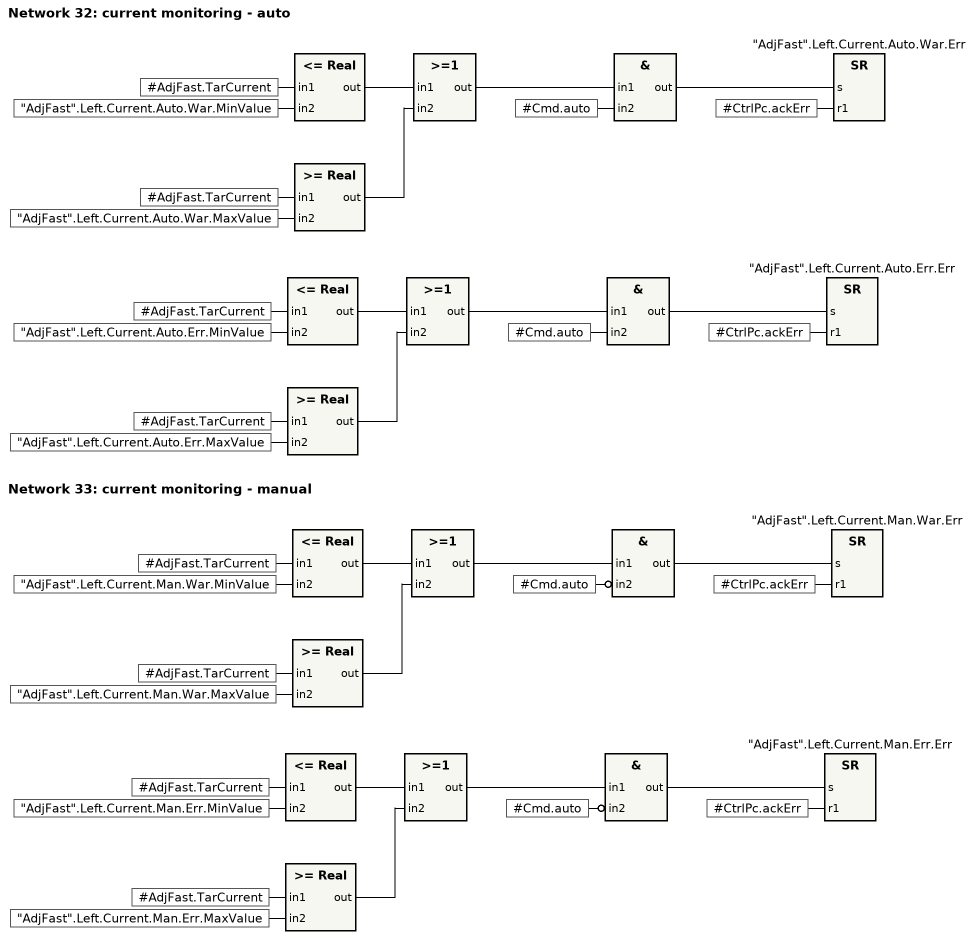
   IF ((#AdjFast.TarCurrent <= "AdjFast".Left.Current.Auto.War.MinValue) OR (#AdjFast.TarCurrent >= "AdjFast".Left.Current.Auto.War.MaxValue)) AND #Cmd.auto THEN
       "AdjFast".Left.Current.Auto.War.Err := TRUE;   // SR flip-flop
   END_IF;
   IF #CtrlPc.ackErr THEN "AdjFast".Left.Current.Auto.War.Err := FALSE; END_IF;
   IF ((#AdjFast.TarCurrent <= "AdjFast".Left.Current.Auto.Err.MinValue) OR (#AdjFast.TarCurrent >= "AdjFast".Left.Current.Auto.Err.MaxValue)) AND #Cmd.auto THEN
       "AdjFast".Left.Current.Auto.Err.Err := TRUE;   // SR flip-flop
   END_IF;
   IF #CtrlPc.ackErr THEN "AdjFast".Left.Current.Auto.Err.Err := FALSE; END_IF;
END_REGION

REGION Network 33: current monitoring - manual
   IF ((#AdjFast.TarCurrent <= "AdjFast".Left.Current.Man.War.MinValue) OR (#AdjFast.TarCurrent >= "AdjFast".Left.Current.Man.War.MaxValue)) AND NOT #Cmd.auto THEN
       "AdjFast".Left.Current.Man.War.Err := TRUE;   // SR flip-flop
   END_IF;
   IF #CtrlPc.ackErr THEN "AdjFast".Left.Current.Man.War.Err := FALSE; END_IF;
   IF ((#AdjFast.TarCurrent <= "AdjFast".Left.Current.Man.Err.MinValue) OR (#AdjFast.TarCurrent >= "AdjFast".Left.Current.Man.Err.MaxValue)) AND NOT #Cmd.auto THEN
       "AdjFast".Left.Current.Man.Err.Err := TRUE;   // SR flip-flop
   END_IF;
   IF #CtrlPc.ackErr THEN "AdjFast".Left.Current.Man.Err.Err := FALSE; END_IF;
END_REGION
END_FUNCTION_BLOCK

FUNCTION_BLOCK "AdjRight"   // FB530, FBD
{ S7_Optimized_Access := 'TRUE' }
// stored: AutoNumber false, MemoryReserve 100, SetENOAutomatically false
   VAR
      Var { ExternalAccessible := 'False'; ExternalVisible := 'False'; ExternalWritable := 'False'} : "TypeVar";
      Cmd { ExternalAccessible := 'False'; ExternalVisible := 'False'; ExternalWritable := 'False'} : "TypeCmd";
      Enc { ExternalAccessible := 'False'; ExternalVisible := 'False'; ExternalWritable := 'False'} : "SysCounterFast";
      Pos { ExternalAccessible := 'False'; ExternalVisible := 'False'; ExternalWritable := 'False'} : "SysPos";
      AdjSlow { ExternalAccessible := 'False'; ExternalVisible := 'False'; ExternalWritable := 'False'} : "SysMotor";
      AdjFast { ExternalAccessible := 'False'; ExternalVisible := 'False'; ExternalWritable := 'False'} : "SysLinMotC1150";
      TAutoOn { ExternalAccessible := 'False'; ExternalVisible := 'False'; ExternalWritable := 'False'} : TON_TIME;
      TAutoTarPosManOn { ExternalAccessible := 'False'; ExternalVisible := 'False'; ExternalWritable := 'False'} : TON_TIME;
      T { ExternalAccessible := 'False'; ExternalVisible := 'False'; ExternalWritable := 'False'} : Array[1..5] of IEC_TIMER;
      adjFastPnSlaveOff { ExternalAccessible := 'False'; ExternalVisible := 'False'; ExternalWritable := 'False'} : "SysPnSlaveDeactivate";
      tarOld { ExternalAccessible := 'False'; ExternalVisible := 'False'; ExternalWritable := 'False'} : DInt;
      autoTarPosMan { ExternalAccessible := 'False'; ExternalVisible := 'False'; ExternalWritable := 'False'} : Bool;
      setValueEnc { ExternalAccessible := 'False'; ExternalVisible := 'False'; ExternalWritable := 'False'} : Bool;
      autoRef { ExternalAccessible := 'False'; ExternalVisible := 'False'; ExternalWritable := 'False'} : Bool;
      posOld { ExternalAccessible := 'False'; ExternalVisible := 'False'; ExternalWritable := 'False'} : Real;
      posDiff { ExternalAccessible := 'False'; ExternalVisible := 'False'; ExternalWritable := 'False'} : Real;
   END_VAR
   VAR_TEMP
      CtrlPc : Struct
         ackErr : Bool;
         manModeActive : Bool;
         manP : Bool;
         manM : Bool;
         manRefRun : Bool;
      END_STRUCT;
      CtrlLinMot : Struct
         mode : Int;
         target : Real;
         speed : Real;
         acc : Real;
         dec : Real;
         jerk : Real;
         autoRef : Bool;
      END_STRUCT;
      refPosDiff : DInt;
      offsetNoStd : Real;
      refPosDiffCalib : DInt;
      modeCalib : Int;
      disMechanicToZero : Int;   // distance mechanic part right to zero [mm]
   END_VAR
   VAR_TEMP   // added for the SCL form of the ladder/FBD networks
      _w1 : Bool;
   END_VAR
BEGIN

REGION Network 1 (SCL): offset for no standard calibration
   (* 
   normally the distance from camera to board should be 550mm
   for special application the distance is different
   the distance can be changed in the goldeneye program
   if its different then 550mm a offset will be added
   *)
   #offsetNoStd := 0.0;
   IF "ComRd".Data.Right.RefPosToBoard <> 550 THEN
       #offsetNoStd := (DINT_TO_REAL("ComRd".Data.Right.RefPosToBoard) - 550.0);
   ELSE
       #offsetNoStd := 0.0;
   END_IF;
END_REGION

REGION Network 2 (SCL): calibration value for offset
   (* 
   modus for calibartion
   camera must be referenced first
   mode 1 -->   the camera must be moved manually to position 550mm from board and
                 then press "Set Nullpoint"
   mode 2 -->   the camera must be moved to a other position and
                 then must be measured from the calibration tool to the camera and
                 this value must be putted in after pressing "Set Nullpoint"
   *)         
   #disMechanicToZero := 870; 
   #modeCalib := 2;
   IF #modeCalib = 1 THEN
       #refPosDiffCalib := "ComRd".Data.Right.TargetPos;
   ELSIF #modeCalib = 2 THEN
       #refPosDiffCalib := (#disMechanicToZero * 10) - ("ComRd".Data.Right.CalibratePos + 5500);
   END_IF;
END_REGION

REGION Network 3 (SCL): calibration value from pc
   "ComSd".Data.Right.SetCalibratePosOk := FALSE;

   IF "ComRd".Data.Right.SetCalibratePos THEN

       IF "G".Cfg.adjRightActive THEN
           #refPosDiff := REAL_TO_DINT("Enc"."8BC1.R".act * 10.0) - #refPosDiffCalib;
       ELSIF "G".Cfg.adjRightActiveLinMot THEN
           #refPosDiff := REAL_TO_DINT("Enc"."8U1.R".act * 10.0) - #refPosDiffCalib;
       END_IF;

       "Ref".adjRightCalOffset := #refPosDiff;
       "ComSd".Data.Right.SetCalibratePosOk := TRUE;

   END_IF;
END_REGION

REGION Network 4 (SCL): target position
   #Cmd.target := "G".Batch.width / 2.0;
   IF "G".Cfg.modeBoardPassing = 1 AND ("G".Cfg.modeDimension = 2 OR "G".Cfg.modeDimension = 4) AND NOT "G".Batch.stdActive THEN
       #Cmd.target := "G".Batch.width / 2.0 + ("G".Batch.widthMeasure - "G".Batch.width);
   END_IF;

   IF "G".Cfg.modeBoardPassing = 3 AND ("G".Cfg.modeDimension = 2 OR "G".Cfg.modeDimension = 4) AND NOT "G".Batch.stdActive THEN
       #Cmd.target :=  "G".Batch.senRightVal;
   END_IF;

   IF #autoTarPosMan THEN
       #Cmd.target := DINT_TO_REAL("ComRd".Data.Right.TargetPos) / 10.0;
   END_IF;

   "Ref".adjRightTar := #Cmd.target + (DINT_TO_REAL("Ref".adjRightCalOffset) / 10.0) + #offsetNoStd - "Enc"."8B1.B".offset;
END_REGION

REGION Network 5 (SCL): data from pc
   IF NOT "G".errComPc THEN
       #CtrlPc.manModeActive := "ComRd".Data.Right.ManModeActive;
       #CtrlPc.manP := "ComRd".Data.Right.ManPlus;
       #CtrlPc.manM := "ComRd".Data.Right.ManMinus;
       #CtrlPc.manRefRun := "ComRd".Data.Right.ManRefRun;
   ELSE
       #CtrlPc.manModeActive := TRUE;
       #CtrlPc.manP := FALSE;
       #CtrlPc.manM := FALSE;
       #CtrlPc.manRefRun := FALSE;
   END_IF;
   #CtrlPc.ackErr := "G".ack;
END_REGION

REGION Network 6: off
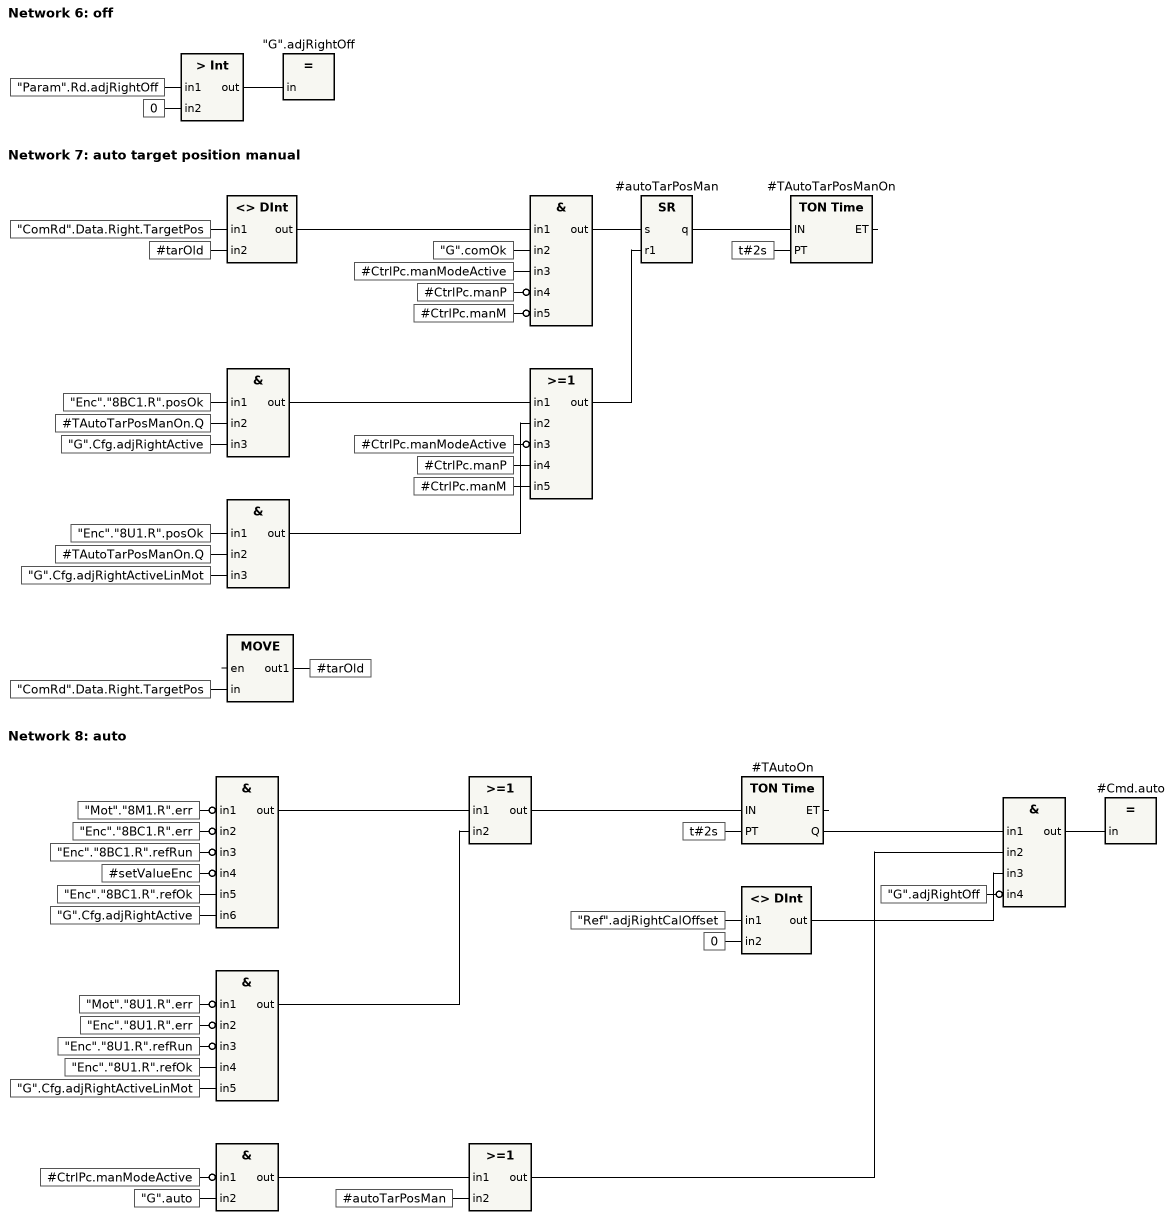
   "G".adjRightOff := "Param".Rd.adjRightOff > 0;
END_REGION

REGION Network 7: auto target position manual
   IF ("ComRd".Data.Right.TargetPos <> #tarOld) AND "G".comOk AND #CtrlPc.manModeActive AND NOT #CtrlPc.manP AND NOT #CtrlPc.manM THEN
       #autoTarPosMan := TRUE;   // SR flip-flop
   END_IF;
   IF ("Enc"."8BC1.R".posOk AND #TAutoTarPosManOn.Q AND "G".Cfg.adjRightActive) OR ("Enc"."8U1.R".posOk AND #TAutoTarPosManOn.Q AND "G".Cfg.adjRightActiveLinMot) OR NOT #CtrlPc.manModeActive OR #CtrlPc.manP OR #CtrlPc.manM THEN
       #autoTarPosMan := FALSE;
   END_IF;
   #TAutoTarPosManOn(IN := #autoTarPosMan, PT := t#2s);   // TON
   #tarOld := "ComRd".Data.Right.TargetPos;
END_REGION

REGION Network 8: auto
   #TAutoOn(IN := (NOT "Mot"."8M1.R".err AND NOT "Enc"."8BC1.R".err AND NOT "Enc"."8BC1.R".refRun AND NOT #setValueEnc AND "Enc"."8BC1.R".refOk AND "G".Cfg.adjRightActive) OR (NOT "Mot"."8U1.R".err AND NOT "Enc"."8U1.R".err AND NOT "Enc"."8U1.R".refRun AND "Enc"."8U1.R".refOk AND "G".Cfg.adjRightActiveLinMot),   // TON
            PT := t#2s);
   #Cmd.auto := #TAutoOn.Q AND ((NOT #CtrlPc.manModeActive AND "G".auto) OR #autoTarPosMan) AND ("Ref".adjRightCalOffset <> 0) AND NOT "G".adjRightOff;
END_REGION

REGION Network 9: manual
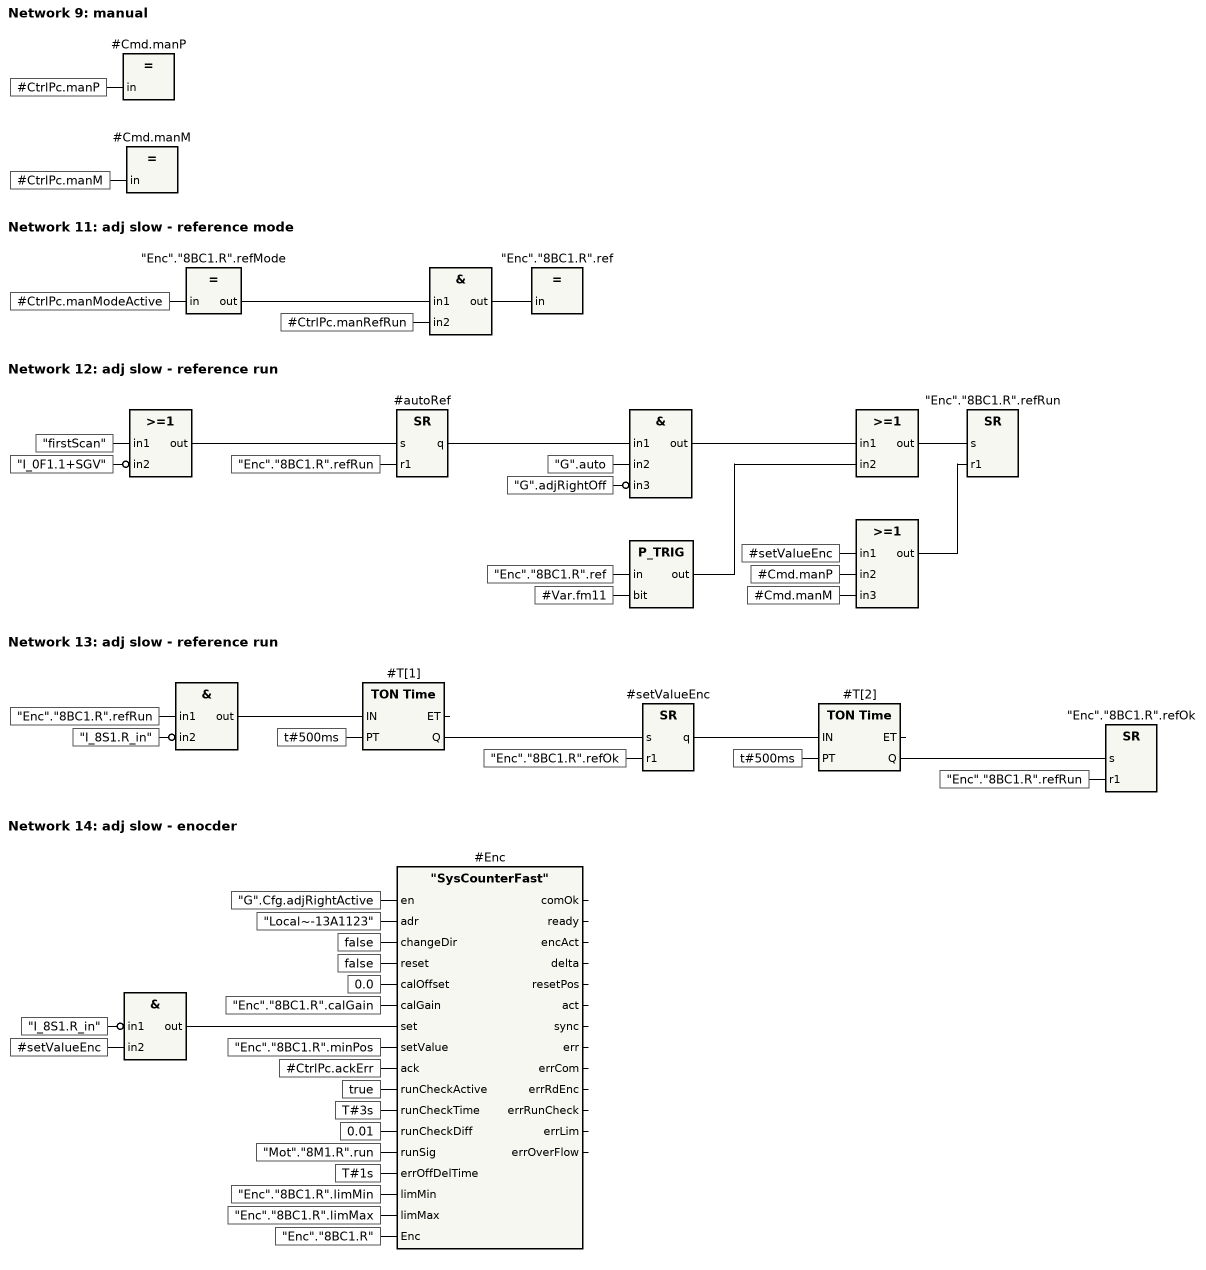
   #Cmd.manP := #CtrlPc.manP;
   #Cmd.manM := #CtrlPc.manM;
END_REGION

REGION Network 10 (SCL): adj slow - calibration value
   "Enc"."8BC1.R".calGain := -0.0275;

   "Enc"."8BC1.R".minPos := 10.0;
   "Enc"."8BC1.R".maxPos := 210.0;

   "Enc"."8BC1.R".limMin := "Enc"."8BC1.R".minPos - 5.0;
   "Enc"."8BC1.R".limMax := "Enc"."8BC1.R".maxPos + 5.0;

   "Enc"."8BC1.R".tarMinPos := "Enc"."8BC1.R".minPos + 0.0;
   "Enc"."8BC1.R".tarMaxPos := "Enc"."8BC1.R".maxPos - 0.0;
END_REGION

REGION Network 11: adj slow - reference mode
   "Enc"."8BC1.R".refMode := #CtrlPc.manModeActive;
   "Enc"."8BC1.R".ref := #CtrlPc.manModeActive AND #CtrlPc.manRefRun;
END_REGION

REGION Network 12: adj slow - reference run
   IF "firstScan" OR NOT "I_0F1.1+SGV" THEN
       #autoRef := TRUE;   // SR flip-flop
   END_IF;
   IF "Enc"."8BC1.R".refRun THEN #autoRef := FALSE; END_IF;
   #_w1 := "Enc"."8BC1.R".ref AND NOT #Var.fm11;   // rising edge
   #Var.fm11 := "Enc"."8BC1.R".ref;
   IF (#autoRef AND "G".auto AND NOT "G".adjRightOff) OR #_w1 THEN
       "Enc"."8BC1.R".refRun := TRUE;   // SR flip-flop
   END_IF;
   IF #setValueEnc OR #Cmd.manP OR #Cmd.manM THEN "Enc"."8BC1.R".refRun := FALSE; END_IF;
END_REGION

REGION Network 13: adj slow - reference run
   #T[1].TON(IN := "Enc"."8BC1.R".refRun AND NOT "I_8S1.R_in", PT := t#500ms);
   IF #T[1].Q THEN
       #setValueEnc := TRUE;   // SR flip-flop
   END_IF;
   IF "Enc"."8BC1.R".refOk THEN #setValueEnc := FALSE; END_IF;
   #T[2].TON(IN := #setValueEnc, PT := t#500ms);
   IF #T[2].Q THEN
       "Enc"."8BC1.R".refOk := TRUE;   // SR flip-flop
   END_IF;
   IF "Enc"."8BC1.R".refRun THEN "Enc"."8BC1.R".refOk := FALSE; END_IF;
END_REGION

REGION Network 14: adj slow - enocder
   IF "G".Cfg.adjRightActive THEN
       #Enc(adr := "Local~-13A1123",   // "SysCounterFast"
            changeDir := false,
            reset := false,
            calOffset := 0.0,
            calGain := "Enc"."8BC1.R".calGain,
            set := NOT "I_8S1.R_in" AND #setValueEnc,
            setValue := "Enc"."8BC1.R".minPos,
            ack := #CtrlPc.ackErr,
            runCheckActive := true,
            runCheckTime := T#3s,
            runCheckDiff := 0.01,
            runSig := "Mot"."8M1.R".run,
            errOffDelTime := T#1s,
            limMin := "Enc"."8BC1.R".limMin,
            limMax := "Enc"."8BC1.R".limMax,
            Enc := "Enc"."8BC1.R");
   END_IF;
END_REGION

REGION Network 15: adj slow - pos
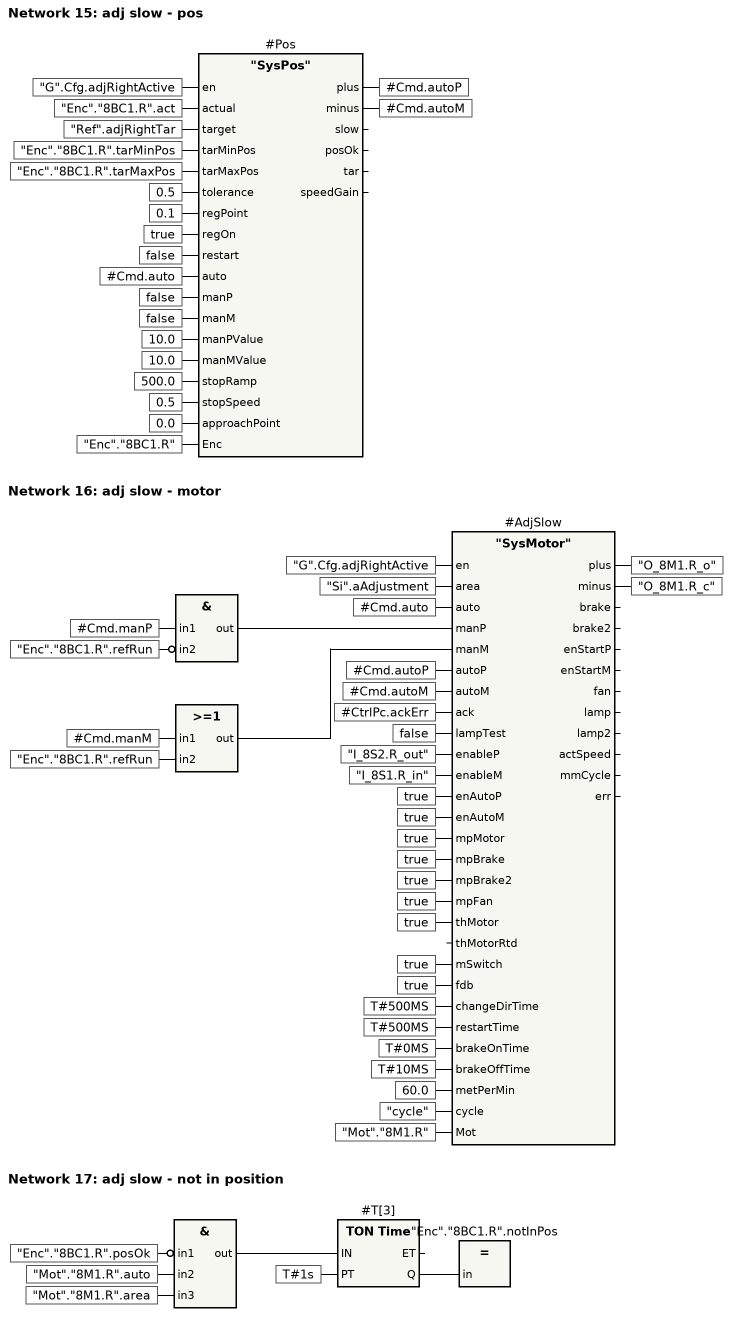
   IF "G".Cfg.adjRightActive THEN
       #Pos(actual := "Enc"."8BC1.R".act,   // "SysPos"
            target := "Ref".adjRightTar,
            tarMinPos := "Enc"."8BC1.R".tarMinPos,
            tarMaxPos := "Enc"."8BC1.R".tarMaxPos,
            tolerance := 0.5,
            regPoint := 0.1,
            regOn := true,
            restart := false,
            auto := #Cmd.auto,
            manP := false,
            manM := false,
            manPValue := 10.0,
            manMValue := 10.0,
            stopRamp := 500.0,
            stopSpeed := 0.5,
            approachPoint := 0.0,
            Enc := "Enc"."8BC1.R",
            plus => #Cmd.autoP,
            minus => #Cmd.autoM);
   END_IF;
END_REGION

REGION Network 16: adj slow - motor
   IF "G".Cfg.adjRightActive THEN
       #AdjSlow(area := "Si".aAdjustment,   // "SysMotor"
                auto := #Cmd.auto,
                manP := #Cmd.manP AND NOT "Enc"."8BC1.R".refRun,
                manM := #Cmd.manM OR "Enc"."8BC1.R".refRun,
                autoP := #Cmd.autoP,
                autoM := #Cmd.autoM,
                ack := #CtrlPc.ackErr,
                lampTest := false,
                enableP := "I_8S2.R_out",
                enableM := "I_8S1.R_in",
                enAutoP := true,
                enAutoM := true,
                mpMotor := true,
                mpBrake := true,
                mpBrake2 := true,
                mpFan := true,
                thMotor := true,
                mSwitch := true,
                fdb := true,
                changeDirTime := T#500MS,
                restartTime := T#500MS,
                brakeOnTime := T#0MS,
                brakeOffTime := T#10MS,
                metPerMin := 60.0,
                cycle := "cycle",
                Mot := "Mot"."8M1.R",
                plus => "O_8M1.R_o",
                minus => "O_8M1.R_c");
   END_IF;
END_REGION

REGION Network 17: adj slow - not in position
   #T[3].TON(IN := NOT "Enc"."8BC1.R".posOk AND "Mot"."8M1.R".auto AND "Mot"."8M1.R".area, PT := T#1s);
   "Enc"."8BC1.R".notInPos := #T[3].Q;
END_REGION

REGION Network 18: adj slow - sensor monitoring
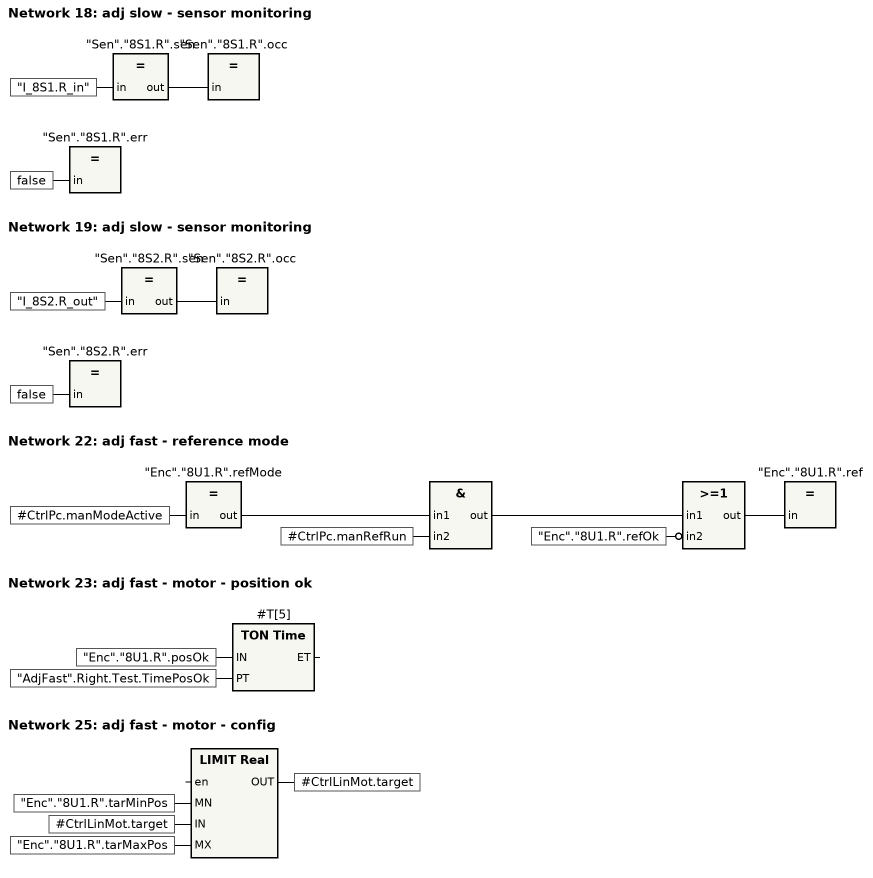
   "Sen"."8S1.R".sen := "I_8S1.R_in";
   "Sen"."8S1.R".occ := "I_8S1.R_in";
   "Sen"."8S1.R".err := false;
END_REGION

REGION Network 19: adj slow - sensor monitoring
   "Sen"."8S2.R".sen := "I_8S2.R_out";
   "Sen"."8S2.R".occ := "I_8S2.R_out";
   "Sen"."8S2.R".err := false;
END_REGION

REGION Network 21 (SCL): adj fast - calibration value
   "Enc"."8U1.R".calGain := 1.0;

   "Enc"."8U1.R".minPos := 5.0;
   "Enc"."8U1.R".maxPos := 155.0;

   "Enc"."8U1.R".limMin := "Enc"."8U1.R".minPos - 5.0;
   "Enc"."8U1.R".limMax := "Enc"."8U1.R".maxPos + 5.0;

   "Enc"."8U1.R".tarMinPos := "Enc"."8U1.R".minPos + 0.0;
   "Enc"."8U1.R".tarMaxPos := "Enc"."8U1.R".maxPos - 0.0;
END_REGION

REGION Network 22: adj fast - reference mode
   "Enc"."8U1.R".refMode := #CtrlPc.manModeActive;
   "Enc"."8U1.R".ref := (#CtrlPc.manModeActive AND #CtrlPc.manRefRun) OR NOT "Enc"."8U1.R".refOk;
END_REGION

REGION Network 23: adj fast - motor - position ok
   #T[5].TON(IN := "Enc"."8U1.R".posOk, PT := "AdjFast".Right.Test.TimePosOk);
END_REGION

REGION Network 24 (SCL): adj fast - motor - config

   //############################################################
   // min            5     mm
   // max          155     mm

   // speed        02      m/s
   // acc/dec      24      m/s2
   // jerk         450     m/s3

   // mode         BestehornVAJ
   //############################################################

   // only testmode for plc
   IF "AdjFast".Right.Test.ModeActive AND NOT #CtrlPc.manModeActive THEN
       IF "AdjFast".Right.Test.TarPos = "AdjFast".Right.Test.TarPos1 AND #T[5].Q THEN
           "AdjFast".Right.Test.TarPos := "AdjFast".Right.Test.TarPos2;
       ELSIF "AdjFast".Right.Test.TarPos = "AdjFast".Right.Test.TarPos2 AND #T[5].Q THEN
           "AdjFast".Right.Test.TarPos := "AdjFast".Right.Test.TarPos1;
       END_IF;
       "Ref".adjRightTar := "AdjFast".Right.Test.TarPos;
   END_IF;

   // active mode
   #CtrlLinMot.mode := 3;
   #CtrlLinMot.target := "Ref".adjRightTar;
   #CtrlLinMot.speed := 2.0;
   #CtrlLinMot.acc := 24.0;
   #CtrlLinMot.dec := 0.0;
   #CtrlLinMot.jerk := 450.0;

   // only testmode for plc
   IF "AdjFast".Right.Mode = 1 THEN
       #CtrlLinMot.mode := 1;
       #CtrlLinMot.target := "AdjFast".Right.VAI.Par1;
       #CtrlLinMot.speed := "AdjFast".Right.VAI.Par2;
       #CtrlLinMot.acc := "AdjFast".Right.VAI.Par3;
       #CtrlLinMot.dec := "AdjFast".Right.VAI.Par4;
       #CtrlLinMot.jerk := 0.0;
   ELSIF "AdjFast".Right.Mode = 2 THEN
       #CtrlLinMot.mode := 2;
       #CtrlLinMot.target := "AdjFast".Right.SinVA.Par1;
       #CtrlLinMot.speed := "AdjFast".Right.SinVA.Par2;
       #CtrlLinMot.acc := "AdjFast".Right.SinVA.Par3;
       #CtrlLinMot.dec := 0.0;
       #CtrlLinMot.jerk := 0.0;
   ELSIF "AdjFast".Right.Mode = 3 THEN
       #CtrlLinMot.mode := 3;
       #CtrlLinMot.target := "AdjFast".Right.BestehornVAJ.Par1;
       #CtrlLinMot.speed := "AdjFast".Right.BestehornVAJ.Par2;
       #CtrlLinMot.acc := "AdjFast".Right.BestehornVAJ.Par3;
       #CtrlLinMot.dec := 0.0;
       #CtrlLinMot.jerk := "AdjFast".Right.BestehornVAJ.Par4;
   END_IF;
END_REGION

REGION Network 25: adj fast - motor - config
   #CtrlLinMot.target := LIMIT(MN := "Enc"."8U1.R".tarMinPos, IN := #CtrlLinMot.target, MX := "Enc"."8U1.R".tarMaxPos);
END_REGION

REGION Network 26: adj fast - motor
   // #CtrlLinMot.target
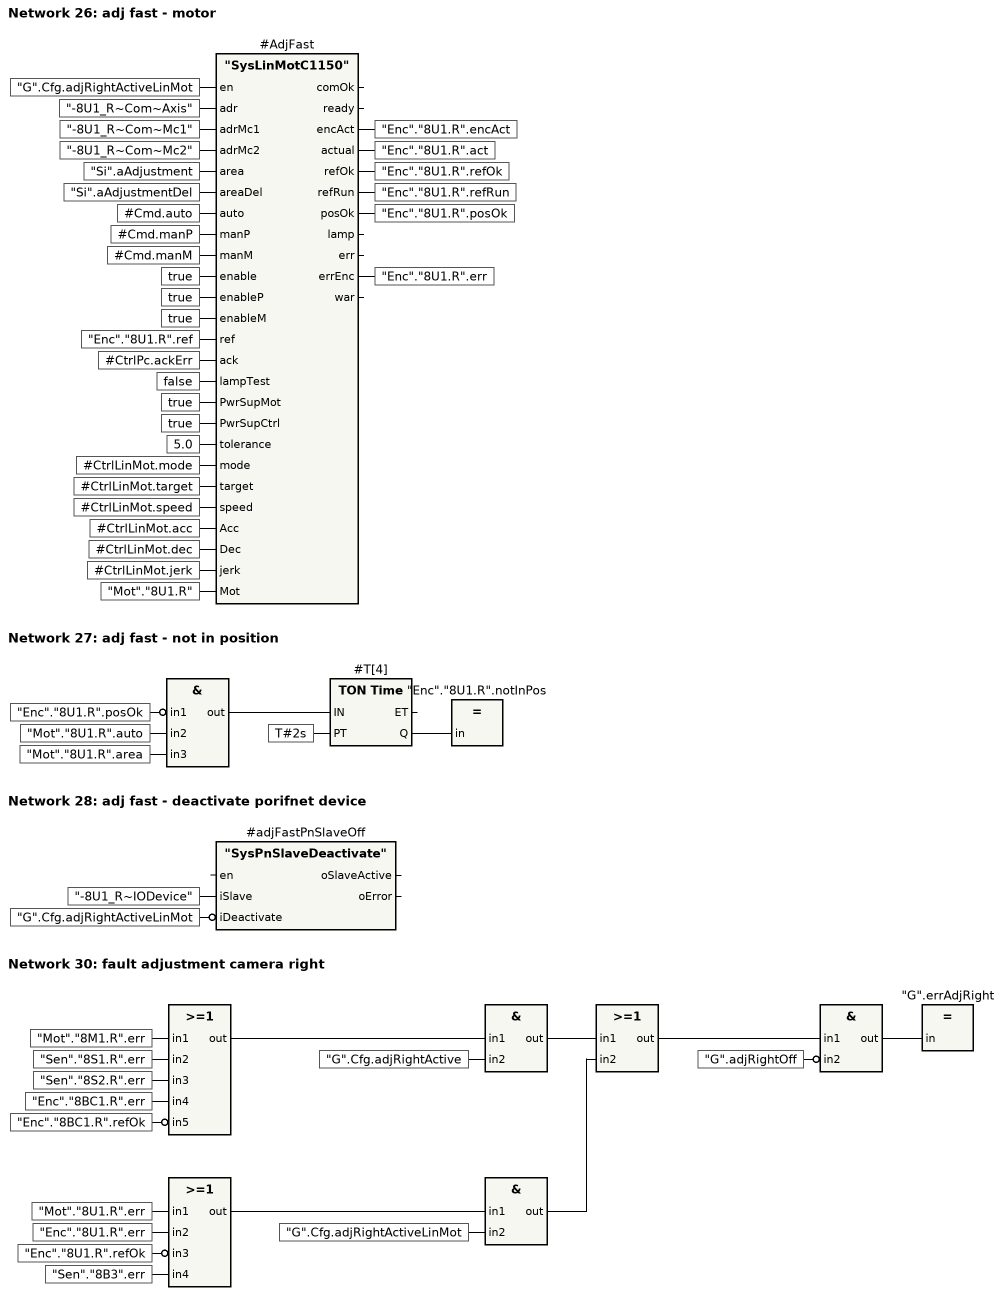
   IF "G".Cfg.adjRightActiveLinMot THEN
       #AdjFast(adr := "-8U1_R~Com~Axis",   // "SysLinMotC1150"
                adrMc1 := "-8U1_R~Com~Mc1",
                adrMc2 := "-8U1_R~Com~Mc2",
                area := "Si".aAdjustment,
                areaDel := "Si".aAdjustmentDel,
                auto := #Cmd.auto,
                manP := #Cmd.manP,
                manM := #Cmd.manM,
                enable := true,
                enableP := true,
                enableM := true,
                ref := "Enc"."8U1.R".ref,
                ack := #CtrlPc.ackErr,
                lampTest := false,
                PwrSupMot := true,
                PwrSupCtrl := true,
                tolerance := 5.0,
                mode := #CtrlLinMot.mode,
                target := #CtrlLinMot.target,
                speed := #CtrlLinMot.speed,
                Acc := #CtrlLinMot.acc,
                Dec := #CtrlLinMot.dec,
                jerk := #CtrlLinMot.jerk,
                Mot := "Mot"."8U1.R",
                encAct => "Enc"."8U1.R".encAct,
                actual => "Enc"."8U1.R".act,
                refOk => "Enc"."8U1.R".refOk,
                refRun => "Enc"."8U1.R".refRun,
                posOk => "Enc"."8U1.R".posOk,
                errEnc => "Enc"."8U1.R".err);
   END_IF;
END_REGION

REGION Network 27: adj fast - not in position
   #T[4].TON(IN := NOT "Enc"."8U1.R".posOk AND "Mot"."8U1.R".auto AND "Mot"."8U1.R".area, PT := T#2s);
   "Enc"."8U1.R".notInPos := #T[4].Q;
END_REGION

REGION Network 28: adj fast - deactivate porifnet device
   #adjFastPnSlaveOff(iSlave := "-8U1_R~IODevice", iDeactivate := NOT "G".Cfg.adjRightActiveLinMot);   // "SysPnSlaveDeactivate"
END_REGION

REGION Network 30: fault adjustment camera right
   "G".errAdjRight := ((("Mot"."8M1.R".err OR "Sen"."8S1.R".err OR "Sen"."8S2.R".err OR "Enc"."8BC1.R".err OR NOT "Enc"."8BC1.R".refOk) AND "G".Cfg.adjRightActive) OR (("Mot"."8U1.R".err OR "Enc"."8U1.R".err OR NOT "Enc"."8U1.R".refOk OR "Sen"."8B3".err) AND "G".Cfg.adjRightActiveLinMot)) AND NOT "G".adjRightOff;
END_REGION

REGION Network 31 (SCL): data to pc
   IF "G".Cfg.adjRightActive THEN
       "Ref".adjRightAct := REAL_TO_DINT("Enc"."8BC1.R".act * 10.0) - "Ref".adjRightCalOffset - REAL_TO_DINT(#offsetNoStd * 10.0);
       "ComSd".Data.Right.ActualEncPos := REAL_TO_DINT("Enc"."8BC1.R".act * 10.0);
       "ComSd".Data.Right.ActualPos :=  "Ref".adjRightAct;
       "ComSd".Data.Right.LimitSwitchMin := "Sen"."8S1.R".sen;
       "ComSd".Data.Right.LimitSwitchMax := "Sen"."8S2.R".sen;
       "ComSd".Data.Right.Err := "Mot"."8M1.R".err;
       "ComSd".Data.Right.ErrEnc := "Enc"."8BC1.R".err;
       "ComSd".Data.Right.PosOk := "Enc"."8BC1.R".posOk;
       "ComSd".Data.Right.Plus := "Mot"."8M1.R".plus;
       "ComSd".Data.Right.Minus := "Mot"."8M1.R".minus;
       "ComSd".Data.Right.refRun := "Enc"."8BC1.R".refRun;
       "ComSd".Data.Right.refOk := "Enc"."8BC1.R".refOk;
   ELSIF  "G".Cfg.adjRightActiveLinMot THEN
       "Ref".adjRightAct := REAL_TO_DINT("Enc"."8U1.R".act * 10.0) - "Ref".adjRightCalOffset - REAL_TO_DINT(#offsetNoStd * 10.0);
       "ComSd".Data.Right.ActualEncPos := REAL_TO_DINT("Enc"."8U1.R".act * 10.0);
       "ComSd".Data.Right.ActualPos :=  "Ref".adjRightAct;
       "ComSd".Data.Right.LimitSwitchMin := TRUE;
       "ComSd".Data.Right.LimitSwitchMax := TRUE;
       "ComSd".Data.Right.Err := "Mot"."8U1.R".err;
       "ComSd".Data.Right.ErrEnc := "Enc"."8U1.R".err;
       "ComSd".Data.Right.PosOk := "Enc"."8U1.R".posOk;
       "ComSd".Data.Right.Plus := "Mot"."8U1.R".plus;
       "ComSd".Data.Right.Minus := "Mot"."8U1.R".minus;
       "ComSd".Data.Right.refRun := "Enc"."8U1.R".refRun;
       "ComSd".Data.Right.refOk := "Enc"."8U1.R".refOk;
   ELSE
       "ComSd".Data.Right.ActualEncPos := 0;
       "ComSd".Data.Right.ActualPos := 0;
       "ComSd".Data.Right.LimitSwitchMin := FALSE;
       "ComSd".Data.Right.LimitSwitchMax := FALSE;
       "ComSd".Data.Right.Err := FALSE;
       "ComSd".Data.Right.ErrEnc := FALSE;
       "ComSd".Data.Right.PosOk := TRUE;
       "ComSd".Data.Right.Plus := FALSE;
       "ComSd".Data.Right.Minus := FALSE;
       "ComSd".Data.Right.refRun := FALSE;
       "ComSd".Data.Right.refOk := TRUE;
   END_IF;
END_REGION

REGION Network 32: current monitoring - auto
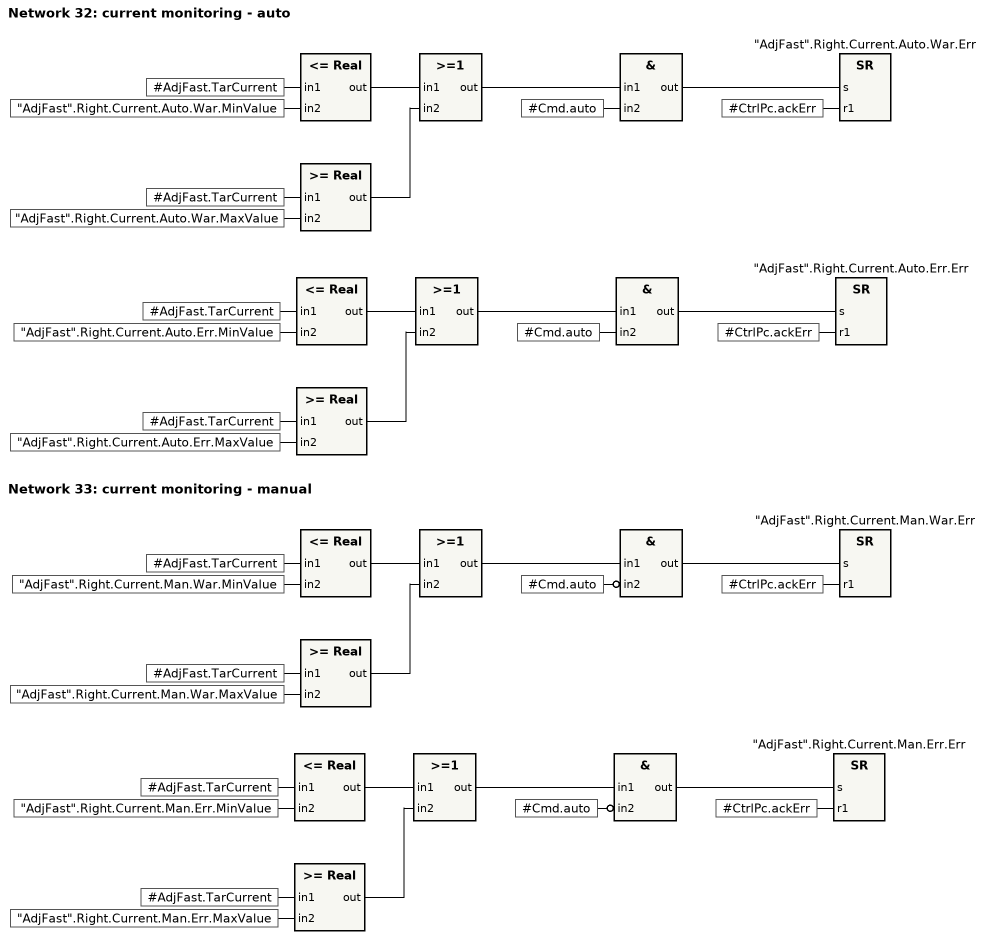
   IF ((#AdjFast.TarCurrent <= "AdjFast".Right.Current.Auto.War.MinValue) OR (#AdjFast.TarCurrent >= "AdjFast".Right.Current.Auto.War.MaxValue)) AND #Cmd.auto THEN
       "AdjFast".Right.Current.Auto.War.Err := TRUE;   // SR flip-flop
   END_IF;
   IF #CtrlPc.ackErr THEN "AdjFast".Right.Current.Auto.War.Err := FALSE; END_IF;
   IF ((#AdjFast.TarCurrent <= "AdjFast".Right.Current.Auto.Err.MinValue) OR (#AdjFast.TarCurrent >= "AdjFast".Right.Current.Auto.Err.MaxValue)) AND #Cmd.auto THEN
       "AdjFast".Right.Current.Auto.Err.Err := TRUE;   // SR flip-flop
   END_IF;
   IF #CtrlPc.ackErr THEN "AdjFast".Right.Current.Auto.Err.Err := FALSE; END_IF;
END_REGION

REGION Network 33: current monitoring - manual
   IF ((#AdjFast.TarCurrent <= "AdjFast".Right.Current.Man.War.MinValue) OR (#AdjFast.TarCurrent >= "AdjFast".Right.Current.Man.War.MaxValue)) AND NOT #Cmd.auto THEN
       "AdjFast".Right.Current.Man.War.Err := TRUE;   // SR flip-flop
   END_IF;
   IF #CtrlPc.ackErr THEN "AdjFast".Right.Current.Man.War.Err := FALSE; END_IF;
   IF ((#AdjFast.TarCurrent <= "AdjFast".Right.Current.Man.Err.MinValue) OR (#AdjFast.TarCurrent >= "AdjFast".Right.Current.Man.Err.MaxValue)) AND NOT #Cmd.auto THEN
       "AdjFast".Right.Current.Man.Err.Err := TRUE;   // SR flip-flop
   END_IF;
   IF #CtrlPc.ackErr THEN "AdjFast".Right.Current.Man.Err.Err := FALSE; END_IF;
END_REGION
END_FUNCTION_BLOCK

FUNCTION_BLOCK "BlowOffValve"   // FB550, FBD
{ S7_Optimized_Access := 'TRUE' }
// stored: AutoNumber false, MemoryReserve 100, SetENOAutomatically false
   VAR
      Var { ExternalAccessible := 'False'; ExternalVisible := 'False'; ExternalWritable := 'False'} : "TypeVar";
      T { ExternalAccessible := 'False'; ExternalVisible := 'False'; ExternalWritable := 'False'} : Array[1..20] of IEC_TIMER;
      blowOff { ExternalAccessible := 'False'; ExternalVisible := 'False'; ExternalWritable := 'False'} : Bool;
      breakTime { ExternalAccessible := 'False'; ExternalVisible := 'False'; ExternalWritable := 'False'} : Time;
      intervallTime { ExternalAccessible := 'False'; ExternalVisible := 'False'; ExternalWritable := 'False'} : Time;
      intervallTimeOff { ExternalAccessible := 'False'; ExternalVisible := 'False'; ExternalWritable := 'False'} : Time;
      bottom { ExternalAccessible := 'False'; ExternalVisible := 'False'; ExternalWritable := 'False'} : Struct
         delayStart : Time;
         Impuls : Time;
         start : Bool;
         blowOff : Bool;
      END_STRUCT;
      left { ExternalAccessible := 'False'; ExternalVisible := 'False'; ExternalWritable := 'False'} : Struct
         delayStart : Time;
         Impuls : Time;
         start : Bool;
         blowOff : Bool;
      END_STRUCT;
      right { ExternalAccessible := 'False'; ExternalVisible := 'False'; ExternalWritable := 'False'} : Struct
         delayStart : Time;
         Impuls : Time;
         start : Bool;
         blowOff : Bool;
      END_STRUCT;
      xray { ExternalAccessible := 'False'; ExternalVisible := 'False'; ExternalWritable := 'False'} : Struct
         delayStart : Time;
         Impuls : Time;
         start : Bool;
         blowOff : Bool;
      END_STRUCT;
   END_VAR
   VAR_TEMP   // added for the SCL form of the ladder/FBD networks
      _w1 : Bool;
   END_VAR
BEGIN

REGION Network 1: pneumatic ok
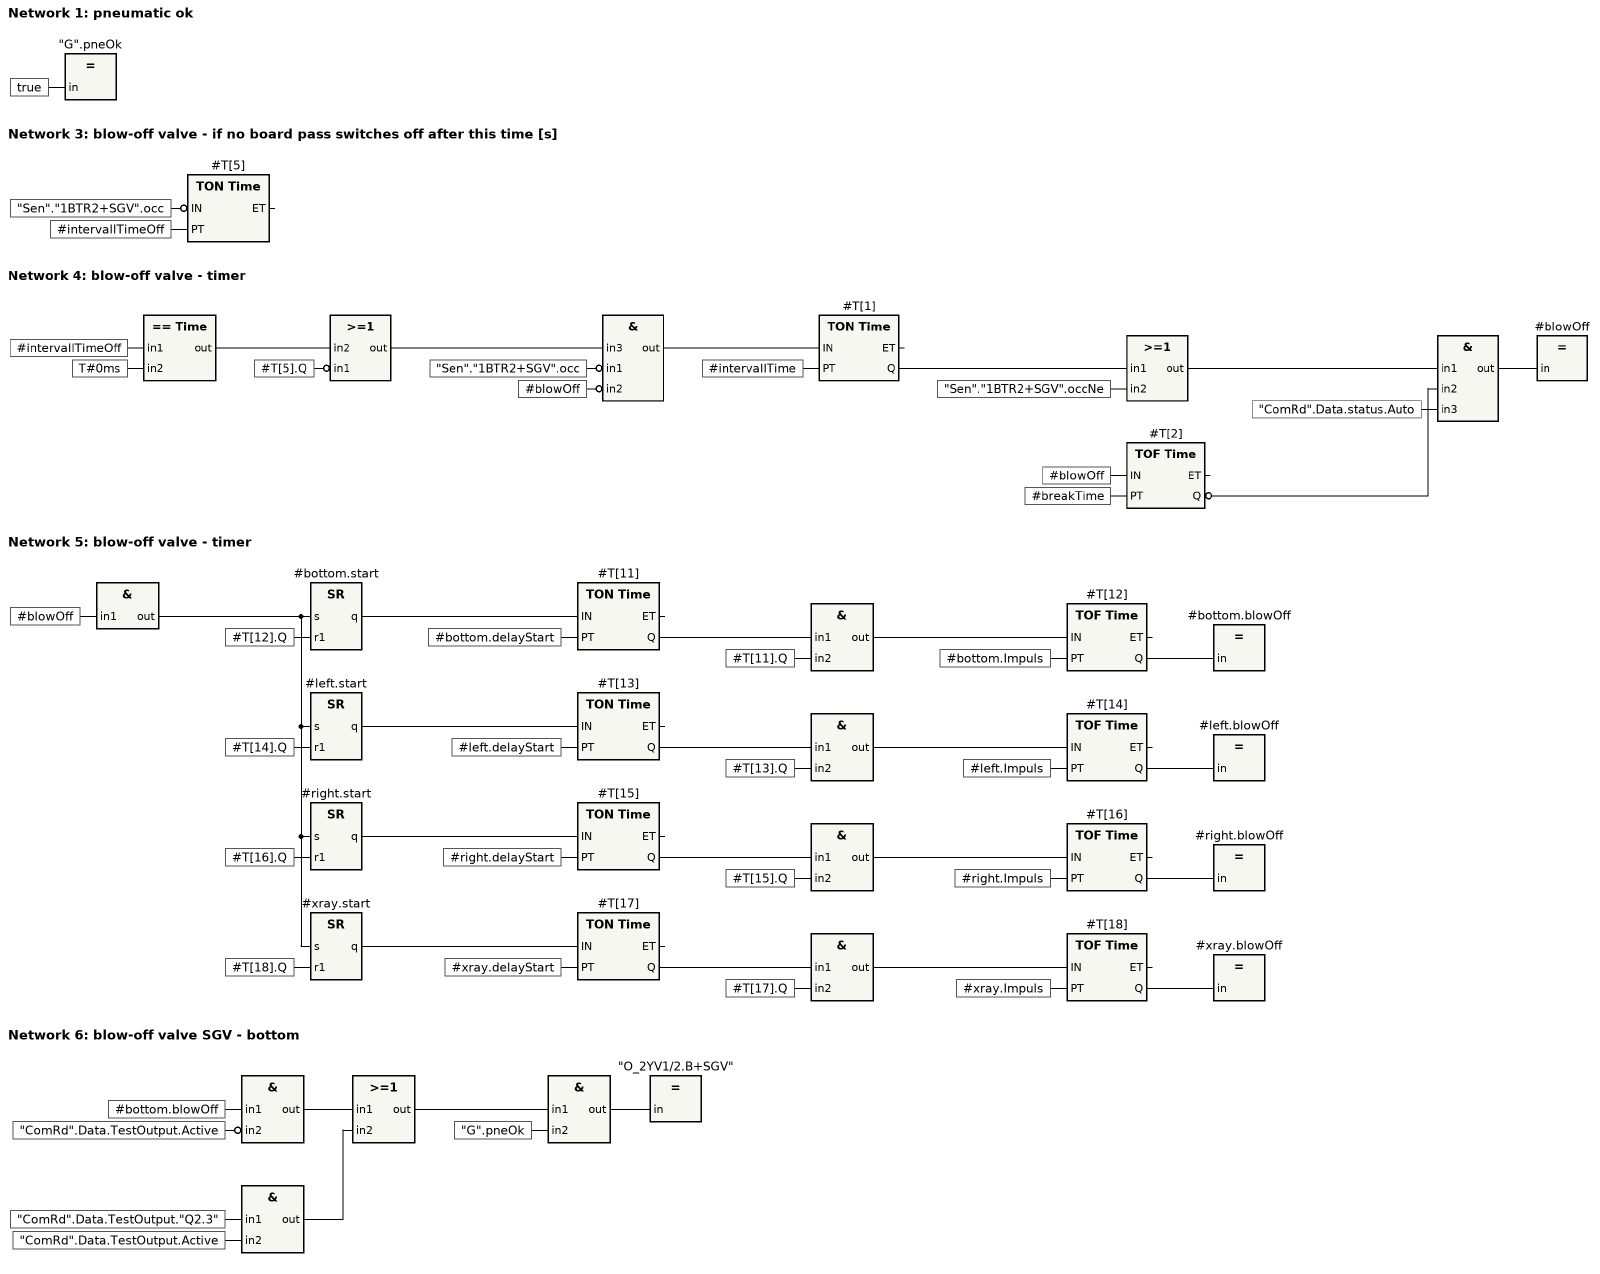
   "G".pneOk := true;
END_REGION

REGION Network 2 (SCL): blow-off valve - parameter

   #breakTime := INT_TO_TIME("Param".Rd.blowOffIbreak);
   #intervallTime := UDINT_TO_TIME(INT_TO_UDINT("Param".Rd.blowOffintervall) * 1000);
   #intervallTimeOff := UDINT_TO_TIME(INT_TO_UDINT("Param".Rd.blowOffintervallOff) * 1000);

   // bottom
   #bottom.delayStart := INT_TO_TIME("Param".Rd.blowOffDelayStartBottom);
   IF "Param".Rd.blowOffImpulsBottom <> 0 THEN
       #bottom.Impuls := INT_TO_TIME("Param".Rd.blowOffImpulsBottom);
   ELSE
       #bottom.Impuls := INT_TO_TIME("Param".Rd.blowOffImpuls);
   END_IF;

   // left
   #left.delayStart := INT_TO_TIME("Param".Rd.blowOffDelayStartLeft);
   IF "Param".Rd.blowOffImpulsLeft <> 0 THEN
       #left.Impuls := INT_TO_TIME("Param".Rd.blowOffImpulsLeft);
   ELSE
       #left.Impuls := INT_TO_TIME("Param".Rd.blowOffImpuls);
   END_IF;

   // right
   #right.delayStart := INT_TO_TIME("Param".Rd.blowOffDelayStartRight);
   IF "Param".Rd.blowOffImpulsRight <> 0 THEN
       #right.Impuls := INT_TO_TIME("Param".Rd.blowOffImpulsRight);
   ELSE
       #right.Impuls := INT_TO_TIME("Param".Rd.blowOffImpuls);
   END_IF;

   // xray
   #xray.delayStart := INT_TO_TIME("Param".Rd.blowOffDelayStartXray);
   IF "Param".Rd.blowOffImpulsXray <> 0 THEN
       #xray.Impuls := INT_TO_TIME("Param".Rd.blowOffImpulsXray);
   ELSE
       #xray.Impuls := INT_TO_TIME("Param".Rd.blowOffImpuls);
   END_IF;
END_REGION

REGION Network 3: blow-off valve - if no board pass switches off after this time [s]
   #T[5].TON(IN := NOT "Sen"."1BTR2+SGV".occ, PT := #intervallTimeOff);
END_REGION

REGION Network 4: blow-off valve - timer
   #T[1].TON(IN := ((#intervallTimeOff = T#0ms) OR NOT #T[5].Q) AND NOT "Sen"."1BTR2+SGV".occ AND NOT #blowOff,
             PT := #intervallTime);
   #_w1 := #T[1].Q OR "Sen"."1BTR2+SGV".occNe;
   #T[2].TOF(IN := #blowOff, PT := #breakTime);
   #blowOff := #_w1 AND NOT #T[2].Q AND "ComRd".Data.status.Auto;
END_REGION

REGION Network 5: blow-off valve - timer
   IF #blowOff THEN
       #bottom.start := TRUE;   // SR flip-flop
   END_IF;
   IF #T[12].Q THEN #bottom.start := FALSE; END_IF;
   #T[11].TON(IN := #bottom.start, PT := #bottom.delayStart);
   #T[12].TOF(IN := #T[11].Q AND #T[11].Q, PT := #bottom.Impuls);
   #bottom.blowOff := #T[12].Q;
   IF #blowOff THEN
       #left.start := TRUE;   // SR flip-flop
   END_IF;
   IF #T[14].Q THEN #left.start := FALSE; END_IF;
   #T[13].TON(IN := #left.start, PT := #left.delayStart);
   #T[14].TOF(IN := #T[13].Q AND #T[13].Q, PT := #left.Impuls);
   #left.blowOff := #T[14].Q;
   IF #blowOff THEN
       #right.start := TRUE;   // SR flip-flop
   END_IF;
   IF #T[16].Q THEN #right.start := FALSE; END_IF;
   #T[15].TON(IN := #right.start, PT := #right.delayStart);
   #T[16].TOF(IN := #T[15].Q AND #T[15].Q, PT := #right.Impuls);
   #right.blowOff := #T[16].Q;
   IF #blowOff THEN
       #xray.start := TRUE;   // SR flip-flop
   END_IF;
   IF #T[18].Q THEN #xray.start := FALSE; END_IF;
   #T[17].TON(IN := #xray.start, PT := #xray.delayStart);
   #T[18].TOF(IN := #T[17].Q AND #T[17].Q, PT := #xray.Impuls);
   #xray.blowOff := #T[18].Q;
END_REGION

REGION Network 6: blow-off valve SGV - bottom
   "O_2YV1/2.B+SGV" := ((#bottom.blowOff AND NOT "ComRd".Data.TestOutput.Active) OR ("ComRd".Data.TestOutput."Q2.3" AND "ComRd".Data.TestOutput.Active)) AND "G".pneOk;
END_REGION

REGION Network 7: blow-off valve SGV - left
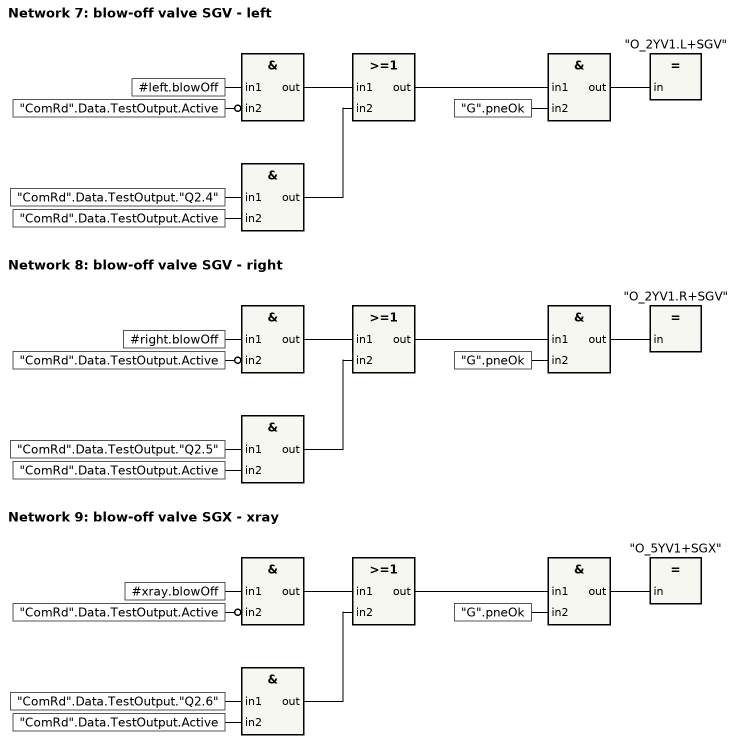
   "O_2YV1.L+SGV" := ((#left.blowOff AND NOT "ComRd".Data.TestOutput.Active) OR ("ComRd".Data.TestOutput."Q2.4" AND "ComRd".Data.TestOutput.Active)) AND "G".pneOk;
END_REGION

REGION Network 8: blow-off valve SGV - right
   "O_2YV1.R+SGV" := ((#right.blowOff AND NOT "ComRd".Data.TestOutput.Active) OR ("ComRd".Data.TestOutput."Q2.5" AND "ComRd".Data.TestOutput.Active)) AND "G".pneOk;
END_REGION

REGION Network 9: blow-off valve SGX - xray
   "O_5YV1+SGX" := ((#xray.blowOff AND NOT "ComRd".Data.TestOutput.Active) OR ("ComRd".Data.TestOutput."Q2.6" AND "ComRd".Data.TestOutput.Active)) AND "G".pneOk;
END_REGION
END_FUNCTION_BLOCK

FUNCTION_BLOCK "AirConditioner"   // FB349, FBD
{ S7_Optimized_Access := 'TRUE' }
// stored: AutoNumber false, MemoryReserve 100, SetENOAutomatically false
   VAR
      Var : "TypeVar";
      T : Array[1..4] of IEC_TIMER;
   END_VAR
   VAR DB_SPECIFIC
      air1Active : Bool := 1;   // air conditioner 1 scannerhousing visual measurement active
      air1InputNo : Bool := 0;   // air conditioner 1 scannerhousing visual measurement input normal
      air2Active : Bool := 1;   // air conditioner 2 scannerhousing visual measurement active
      air2InputNo : Bool := 0;   // air conditioner 2 scannerhousing visual measurement input normal
      airXrayActive : Bool := 1;   // air conditioner scannerhousing x-ray measurement active
      airXrayInputNo : Bool := 0;   // air conditioner scannerhousing x-ray measurement input normal
      airDehActive : Bool := 0;   // air dehumidifier active
      airDehInputNo : Bool := 0;   // air dehumidifier input normal open
   END_VAR
BEGIN

REGION Network 1 (SCL): air conditioner 1&2 visual measurement - config from Pc
   "G".air1Off := INT_TO_BOOL( "Param".Rd.air1Off);
   "G".air2Off := INT_TO_BOOL("Param".Rd.air2Off);
   #air1Active := INT_TO_BOOL("Param".Rd.air1Active);
   #air2Active := INT_TO_BOOL("Param".Rd.air2Active);
   #air1InputNo := INT_TO_BOOL("Param".Rd.air1InputNo);
   #air2InputNo := INT_TO_BOOL("Param".Rd.air2InputNo);
END_REGION

REGION Network 2: air conditioner 1&2 visual measurement - fault
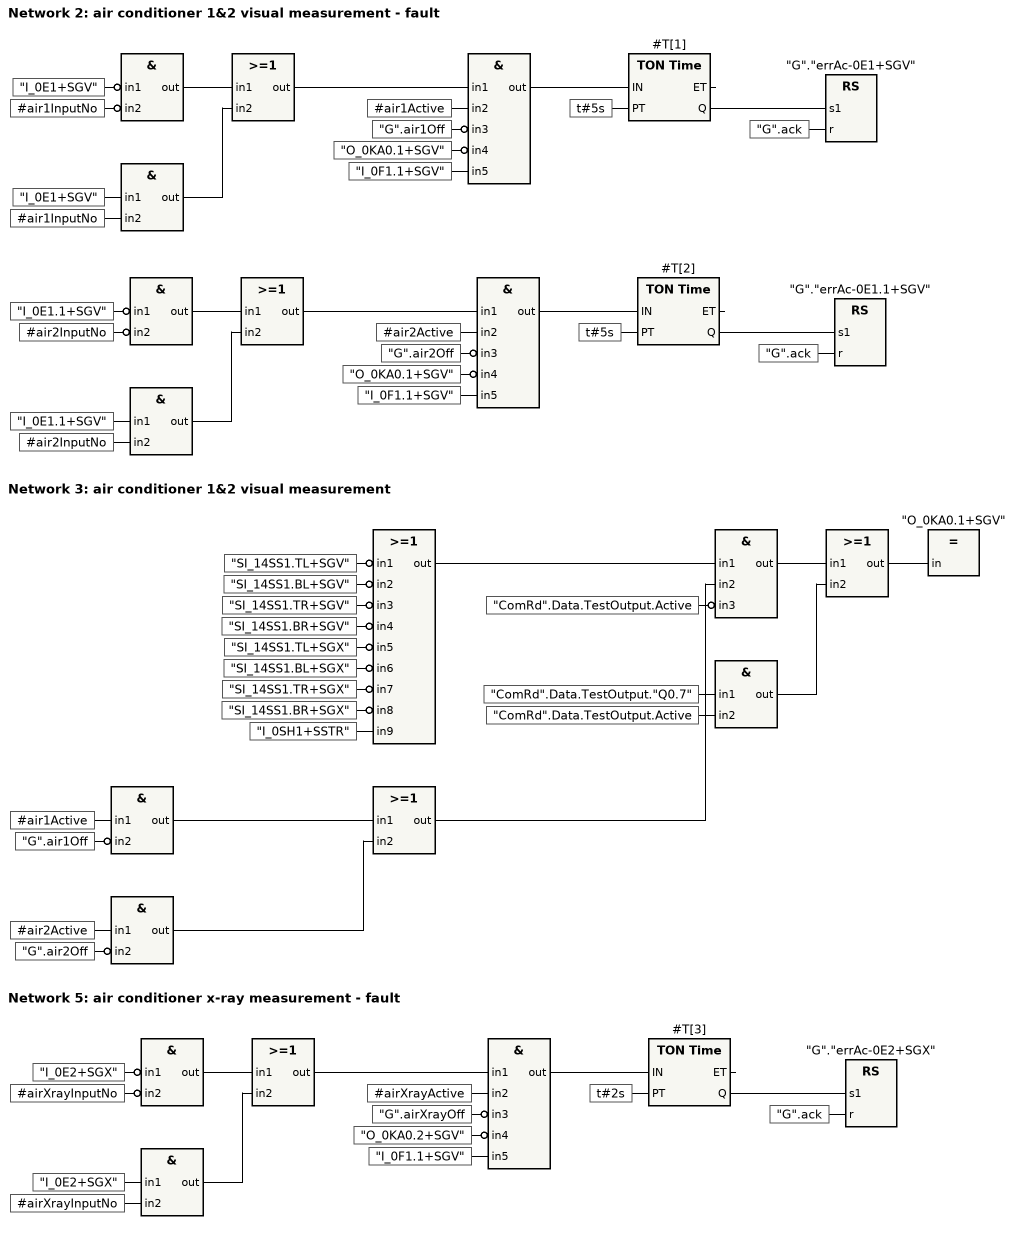
   #T[1].TON(IN := ((NOT "I_0E1+SGV" AND NOT #air1InputNo) OR ("I_0E1+SGV" AND #air1InputNo)) AND #air1Active AND NOT "G".air1Off AND NOT "O_0KA0.1+SGV" AND "I_0F1.1+SGV",
             PT := t#5s);
   IF "G".ack THEN
       "G"."errAc-0E1+SGV" := FALSE;   // RS flip-flop
   END_IF;
   IF #T[1].Q THEN "G"."errAc-0E1+SGV" := TRUE; END_IF;
   #T[2].TON(IN := ((NOT "I_0E1.1+SGV" AND NOT #air2InputNo) OR ("I_0E1.1+SGV" AND #air2InputNo)) AND #air2Active AND NOT "G".air2Off AND NOT "O_0KA0.1+SGV" AND "I_0F1.1+SGV",
             PT := t#5s);
   IF "G".ack THEN
       "G"."errAc-0E1.1+SGV" := FALSE;   // RS flip-flop
   END_IF;
   IF #T[2].Q THEN "G"."errAc-0E1.1+SGV" := TRUE; END_IF;
END_REGION

REGION Network 3: air conditioner 1&2 visual measurement
   "O_0KA0.1+SGV" := ((NOT "SI_14SS1.TL+SGV" OR NOT "SI_14SS1.BL+SGV" OR NOT "SI_14SS1.TR+SGV" OR NOT "SI_14SS1.BR+SGV" OR NOT "SI_14SS1.TL+SGX" OR NOT "SI_14SS1.BL+SGX" OR NOT "SI_14SS1.TR+SGX" OR NOT "SI_14SS1.BR+SGX" OR "I_0SH1+SSTR") AND ((#air1Active AND NOT "G".air1Off) OR (#air2Active AND NOT "G".air2Off)) AND NOT "ComRd".Data.TestOutput.Active) OR ("ComRd".Data.TestOutput."Q0.7" AND "ComRd".Data.TestOutput.Active);
END_REGION

REGION Network 4 (SCL): air conditioner x-ray measurement - config from Pc
   "G".airXrayOff := INT_TO_BOOL( "Param".Rd.airXrayOff);
   #airXrayActive := INT_TO_BOOL("Param".Rd.airXrayActive);
   #airXrayInputNo := INT_TO_BOOL("Param".Rd.airXrayInputNo);
END_REGION

REGION Network 5: air conditioner x-ray measurement - fault
   #T[3].TON(IN := ((NOT "I_0E2+SGX" AND NOT #airXrayInputNo) OR ("I_0E2+SGX" AND #airXrayInputNo)) AND #airXrayActive AND NOT "G".airXrayOff AND NOT "O_0KA0.2+SGV" AND "I_0F1.1+SGV",
             PT := t#2s);
   IF "G".ack THEN
       "G"."errAc-0E2+SGX" := FALSE;   // RS flip-flop
   END_IF;
   IF #T[3].Q THEN "G"."errAc-0E2+SGX" := TRUE; END_IF;
END_REGION

REGION Network 6: air conditioner x-ray measurement - fault
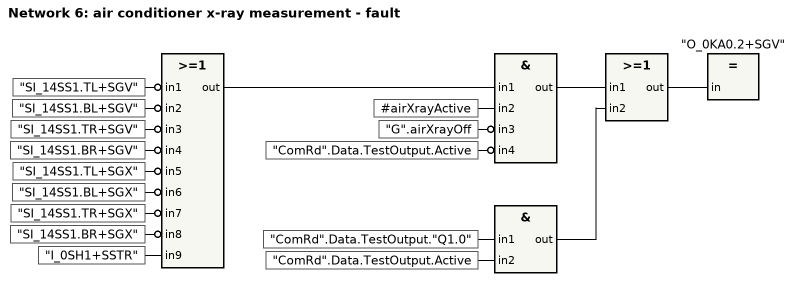
   "O_0KA0.2+SGV" := ((NOT "SI_14SS1.TL+SGV" OR NOT "SI_14SS1.BL+SGV" OR NOT "SI_14SS1.TR+SGV" OR NOT "SI_14SS1.BR+SGV" OR NOT "SI_14SS1.TL+SGX" OR NOT "SI_14SS1.BL+SGX" OR NOT "SI_14SS1.TR+SGX" OR NOT "SI_14SS1.BR+SGX" OR "I_0SH1+SSTR") AND #airXrayActive AND NOT "G".airXrayOff AND NOT "ComRd".Data.TestOutput.Active) OR ("ComRd".Data.TestOutput."Q1.0" AND "ComRd".Data.TestOutput.Active);
END_REGION
END_FUNCTION_BLOCK

ORGANIZATION_BLOCK "Cyclic interrupt 1,5s"   // OB30, FBD, CyclicInterrupt
{ S7_Optimized_Access := 'TRUE' }
// stored: SetENOAutomatically false
   VAR_INPUT
      Initial_Call : Bool;   // Initial call of this OB
      Event_Count : Int;   // Events discarded
   END_VAR
BEGIN

NETWORK
TITLE = call diagnose
      CALL  "Diag", "Diag_DB";

END_ORGANIZATION_BLOCK

FUNCTION_BLOCK "Diag"   // FB60, FBD
TITLE = diagnose
{ S7_Optimized_Access := 'TRUE' }
// stored: AutoNumber false, MemoryReserve 100, SetENOAutomatically false
   VAR
      Var { ExternalAccessible := 'False'; ExternalVisible := 'False'; ExternalWritable := 'False'} : "TypeVar";
      Plc { ExternalAccessible := 'False'; ExternalVisible := 'False'; ExternalWritable := 'False'} : "Diag_PLCCheck";
      PlcData { ExternalAccessible := 'False'; ExternalVisible := 'False'; ExternalWritable := 'False'} : "UserDiag_typePLC";   // PLC diagnostics data
      IoSys1 { ExternalAccessible := 'False'; ExternalVisible := 'False'; ExternalWritable := 'False'} : "Diag_IOSystemCheck";
      IoDataSys1 { ExternalAccessible := 'False'; ExternalVisible := 'False'; ExternalWritable := 'False'} : "UserDiag_typeIOSystem";   // IO-System diagnostics data
   END_VAR
BEGIN

REGION Network 1: Call startup and diagnostics of PLC
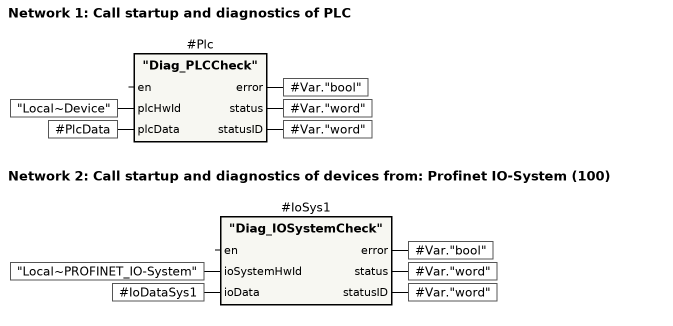
   #Plc(plcHwId := "Local~Device",   // "Diag_PLCCheck"
        plcData := #PlcData,
        error => #Var."bool",
        status => #Var."word",
        statusID => #Var."word");
END_REGION

REGION Network 2: Call startup and diagnostics of devices from: Profinet IO-System (100)
   #IoSys1(ioSystemHwId := "Local~PROFINET_IO-System",   // "Diag_IOSystemCheck"
           ioData := #IoDataSys1,
           error => #Var."bool",
           status => #Var."word",
           statusID => #Var."word");
END_REGION
END_FUNCTION_BLOCK

ORGANIZATION_BLOCK "Diagnostic error interrupt"   // OB82, FBD, DiagnosticErrorInterrupt
{ S7_Optimized_Access := 'TRUE' }
// stored: SetENOAutomatically false
   VAR_INPUT
      IO_State : Word;   // IO state of the HW object
      LADDR : HW_ANY;   // Hardware identifier
      Channel : UInt;   // Channel number
      MultiError : Bool;   // =true if more than one error is present
   END_VAR
BEGIN

NETWORK
TITLE = call diagnose
      CALL  "Diag", "Diag_DB";

END_ORGANIZATION_BLOCK

ORGANIZATION_BLOCK "IO access error"   // OB122, FBD, IOAccessError
{ S7_Optimized_Access := 'TRUE' }
// stored: SetENOAutomatically false
   VAR_INPUT
      BlockNr : UInt;   // Number of causing block
      Reaction : USInt;   // 0:ignore, 1:substitute, 2:skip
      Fault_ID : Byte;   // 16#42:reading, 16#43:writing
      BlockType : USInt;   // 16#01:OB, 16#02:FC, 16#03:FB, 16#04:SFC, 16#05:SFB, 16#06:DB: Type of block causing the error
      Area : USInt;   // 16#81:I, 16#82:Q: IO area where the IOaccess error occured
      DBNr : DB_ANY;   // Reserved for system
      Csg_OBNr : OB_ANY;   // Number of OB causing the error
      Csg_Prio : USInt;   // Priority of OB causing the error
      Width : USInt;   // 0:bit, 1:byte, 2:word, 3:dword, 4:lword
   END_VAR
BEGIN
END_ORGANIZATION_BLOCK

ORGANIZATION_BLOCK "Programming error"   // OB121, FBD, ProgrammingError
{ S7_Optimized_Access := 'TRUE' }
// stored: SetENOAutomatically false
   VAR_INPUT
      BlockNr : UInt;   // Number of causing block
      Reaction : USInt;   // 0:ignore, 1:substitute, 2:skip
      Fault_ID : Byte;   // Fault identifier
      BlockType : USInt;   // 16#01:OB, 16#02:FC, 16#03:FB, 16#04:SFC, 16#05:SFB, 16#06:DB: Type of block causing the error
      Area : USInt;   // Area where the error occured
      DBNr : DB_ANY;   // DB number if Area = DB or DI
      Csg_OBNr : OB_ANY;   // Number of OB causing the error
      Csg_Prio : USInt;   // Priority of OB causing the error
      Width : USInt;   // 0:bit, 1:byte, 2:word, 3:dword, 4:lword
   END_VAR
BEGIN
END_ORGANIZATION_BLOCK

ORGANIZATION_BLOCK "Pull or plug of modules"   // OB83, FBD, PullOrPlugOfModules
{ S7_Optimized_Access := 'TRUE' }
// stored: SetENOAutomatically false
   VAR_INPUT
      LADDR : HW_IO;   // Hardware identifier
      Event_Class : Byte;   // 16#38/39: module inserted, removed
      Fault_ID : Byte;   // Fault identifier
   END_VAR
BEGIN

NETWORK
TITLE = call diagnose
      CALL  "Diag", "Diag_DB";

END_ORGANIZATION_BLOCK

ORGANIZATION_BLOCK "Rack or station failure"   // OB86, FBD, RackOrStationFailure
{ S7_Optimized_Access := 'TRUE' }
// stored: SetENOAutomatically false
   VAR_INPUT
      LADDR : HW_DEVICE;   // Hardware identifier
      Event_Class : Byte;   // Event class
      Fault_ID : Byte;   // Fault identifier
   END_VAR
BEGIN

NETWORK
TITLE = call diagnose
      CALL  "Diag", "Diag_DB";

END_ORGANIZATION_BLOCK

ORGANIZATION_BLOCK "Startup"   // OB100, FBD, Startup
TITLE = "Complete Restart"
{ S7_Optimized_Access := 'TRUE' }
// stored: SetENOAutomatically false
   VAR_INPUT
      LostRetentive : Bool;   // True if retentive data are lost
      LostRTC : Bool;   // True if date and time are lost
   END_VAR
BEGIN

NETWORK
TITLE = first scan
      SET;
      S     "firstScan";

NETWORK
TITLE = call diagnose
      CALL  "Diag", "Diag_DB";

END_ORGANIZATION_BLOCK

ORGANIZATION_BLOCK "Time error interrupt"   // OB80, FBD, TimeErrorInterrupt
{ S7_Optimized_Access := 'TRUE' }
// stored: SetENOAutomatically false
   VAR_INPUT
      Fault_ID : Byte;   // Fault identifier
      Csg_OBnr : OB_ANY;   // Number of OB causing the error
      Csg_Prio : UInt;   // Priority of OB causing the error
   END_VAR
BEGIN
END_ORGANIZATION_BLOCK

FUNCTION_BLOCK "SysFlipFlop"   // FB2000, FBD
TITLE = flip flop used for manual mode/push buttons
{ S7_Optimized_Access := 'TRUE' }
AUTHOR : MiCROTEC
VERSION : 1.0
// -2017.03 : Martin
// stored: AutoNumber false, MemoryReserve 100, SetENOAutomatically false
   VAR_INPUT
      input { ExternalAccessible := 'False'; ExternalVisible := 'False'; ExternalWritable := 'False'} : Bool;   // input toggle
      set { ExternalAccessible := 'False'; ExternalVisible := 'False'; ExternalWritable := 'False'} : Bool;   // set
      reset { ExternalAccessible := 'False'; ExternalVisible := 'False'; ExternalWritable := 'False'} : Bool;   // reset
      lmBlink { ExternalAccessible := 'False'; ExternalVisible := 'False'; ExternalWritable := 'False'} : Bool;   // let blink lamp
      lampTest { ExternalAccessible := 'False'; ExternalVisible := 'False'; ExternalWritable := 'False'} : Bool;   // lamp test
      resetMode { ExternalAccessible := 'False'; ExternalVisible := 'False'; ExternalWritable := 'False'} : Bool;   // 1=output will reset with rising edge from "LmBlink"
      hmiPageTar { ExternalAccessible := 'False'; ExternalVisible := 'False'; ExternalWritable := 'False'} : Int;   // number from hmi Page to open with rising edge from OutSignal
   END_VAR
   VAR_OUTPUT
      out { ExternalAccessible := 'False'; ExternalVisible := 'False'; ExternalWritable := 'False'} : Bool;   // output
      lamp { ExternalAccessible := 'False'; ExternalVisible := 'False'; ExternalWritable := 'False'} : Bool;   // lamp
      lamp2 { ExternalAccessible := 'False'; ExternalVisible := 'False'; ExternalWritable := 'False'} : Bool;   // lamp 2
      lamp3 { ExternalAccessible := 'False'; ExternalVisible := 'False'; ExternalWritable := 'False'} : Bool;   // lamp 3
   END_VAR
   VAR_IN_OUT
      hmiPageAct { ExternalAccessible := 'False'; ExternalVisible := 'False'; ExternalWritable := 'False'} : Int;
   END_VAR
   VAR RETAIN
      ff { ExternalAccessible := 'False'; ExternalVisible := 'False'; ExternalWritable := 'False'} : Bool;
      fl1 { ExternalAccessible := 'False'; ExternalVisible := 'False'; ExternalWritable := 'False'} : Bool;
      fl2 { ExternalAccessible := 'False'; ExternalVisible := 'False'; ExternalWritable := 'False'} : Bool;
      StatOut { ExternalAccessible := 'False'; ExternalVisible := 'False'; ExternalWritable := 'False'} : Bool;   // Setzen Rücksetzen über OP
   END_VAR
   VAR_TEMP   // added for the SCL form of the ladder/FBD networks
      _w1 : Bool;
   END_VAR
BEGIN

REGION Network 1: output
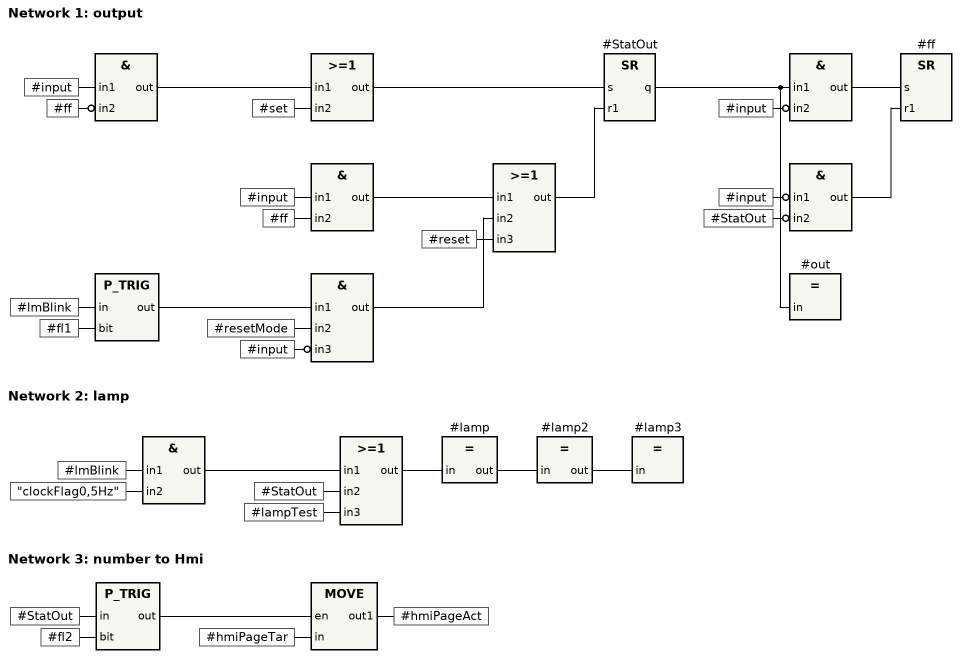
   #_w1 := #lmBlink AND NOT #fl1;   // rising edge
   #fl1 := #lmBlink;
   IF (#input AND NOT #ff) OR #set THEN
       #StatOut := TRUE;   // SR flip-flop
   END_IF;
   IF (#input AND #ff) OR (#_w1 AND #resetMode AND NOT #input) OR #reset THEN #StatOut := FALSE; END_IF;
   IF #StatOut AND NOT #input THEN
       #ff := TRUE;   // SR flip-flop
   END_IF;
   IF NOT #input AND NOT #StatOut THEN #ff := FALSE; END_IF;
   #out := #StatOut;
END_REGION

REGION Network 2: lamp
   #lamp := (#lmBlink AND "clockFlag0,5Hz") OR #StatOut OR #lampTest;
   #lamp2 := #lamp;
   #lamp3 := #lamp;
END_REGION

REGION Network 3: number to Hmi
   #_w1 := #StatOut AND NOT #fl2;   // rising edge
   #fl2 := #StatOut;
   IF #_w1 THEN #hmiPageAct := #hmiPageTar; END_IF;
END_REGION
END_FUNCTION_BLOCK

FUNCTION_BLOCK "ErrComTextList"   // FB305, FBD
{ S7_Optimized_Access := 'TRUE' }
// stored: AutoNumber false, MemoryReserve 100, SetENOAutomatically false
   VAR
      Var { ExternalAccessible := 'False'; ExternalVisible := 'False'; ExternalWritable := 'False'} : "TypeVar";
      T { ExternalAccessible := 'False'; ExternalVisible := 'False'; ExternalWritable := 'False'} : Array[1..3] of IEC_TIMER;
      iLang { ExternalAccessible := 'False'; ExternalVisible := 'False'; ExternalWritable := 'False'} : Array[1..3] of DInt;
      sendImp { ExternalAccessible := 'False'; ExternalVisible := 'False'; ExternalWritable := 'False'} : Bool;
      sendTime { ExternalAccessible := 'False'; ExternalVisible := 'False'; ExternalWritable := 'False'} : Real;
      errNr { ExternalAccessible := 'False'; ExternalVisible := 'False'; ExternalWritable := 'False'} : DInt;
   END_VAR
   VAR_TEMP
      i : DInt;
      i2 : DInt;
      lowBound : DInt;
      upBound : DInt;
   END_VAR
BEGIN

REGION Network 1: sending impulse/clock
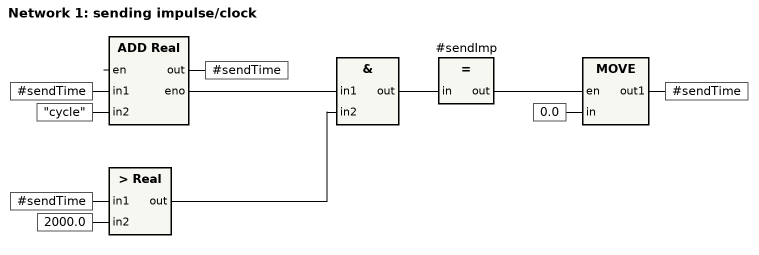
   #sendTime := #sendTime + "cycle";
   #sendImp := #sendTime > 2000.0;
   IF #sendImp THEN #sendTime := 0.0; END_IF;
END_REGION

REGION Network 2 (SCL): send step by step all the error list to Pc
   #lowBound := 2000;
   #upBound := 2205;

   IF #sendImp THEN

       #errNr += 1;
       IF #errNr > #upBound OR #errNr < #lowBound THEN
           #errNr := #lowBound;
       END_IF;

       "ComErrText".Sd.errList.idProd := 0;
       "ComErrText".Sd.errList.id := DINT_TO_UINT(#errNr);
       "ComErrText".Sd.errList.prio := "ErrTextList".err[#errNr].prio;
       "ComErrText".Sd.errList.timeStamp := DT_TO_LDT("Hmi".Clock.Act);

       #iLang[1] := #iLang[2] := #iLang[3] := 1;
       FOR #i := 1 TO 3 DO
           FOR #i2 := 1 TO 8 DO
               IF "ComErrText".Rd.language[#i] = "ErrTextList".language[#i2] AND "ComErrText".Rd.language[#i] <> WSTRING#'' THEN
                   #iLang[#i] := #i2;
                   EXIT;
               END_IF;
           END_FOR;
       END_FOR;

       "ComErrText".Sd.errList.alarm[1] := "ErrTextList".err[#errNr].alarm[#iLang[1]];
       "ComErrText".Sd.errList.info[1] := wstring#'';  
       "ComErrText".Sd.errList.remedy[1] := wstring#'';

       "ComErrText".Sd.errList.alarm[2] := "ErrTextList".err[#errNr].alarm[#iLang[2]];
       "ComErrText".Sd.errList.info[2] := wstring#'';
       "ComErrText".Sd.errList.remedy[2] := wstring#'';

       "ComErrText".Sd.errList.alarm[3] := "ErrTextList".err[#errNr].alarm[#iLang[3]];
       "ComErrText".Sd.errList.info[3] := wstring#'';
       "ComErrText".Sd.errList.remedy[3] := wstring#'';

   END_IF;
END_REGION
END_FUNCTION_BLOCK

DATA_BLOCK "AdjLeft_DB"   // DB525
// stored: AutoNumber false, InstanceOfName AdjLeft, InstanceOfType FB
"AdjLeft"
BEGIN
END_DATA_BLOCK

DATA_BLOCK "AdjRight_DB"   // DB530
// stored: AutoNumber false, InstanceOfName AdjRight, InstanceOfType FB
"AdjRight"
BEGIN
END_DATA_BLOCK

DATA_BLOCK "AdjScanner_DB"   // DB510
// stored: AutoNumber false, InstanceOfName AdjScanner, InstanceOfType FB
"AdjScanner"
BEGIN
END_DATA_BLOCK

DATA_BLOCK "AdjTop_DB"   // DB520
// stored: AutoNumber false, InstanceOfName AdjTop, InstanceOfType FB
"AdjTop"
BEGIN
END_DATA_BLOCK

DATA_BLOCK "AirConditioner_DB"   // DB549
// stored: AutoNumber false, InstanceOfName AirConditioner, InstanceOfType FB
"AirConditioner"
BEGIN
END_DATA_BLOCK

DATA_BLOCK "AutoIndication_DB"   // DB300
// stored: AutoNumber false, InstanceOfName AutoIndication, InstanceOfType FB
"AutoIndication"
BEGIN
END_DATA_BLOCK

DATA_BLOCK "BlowOffValve_DB"   // DB550
// stored: AutoNumber false, InstanceOfName BlowOffValve, InstanceOfType FB
"BlowOffValve"
BEGIN
END_DATA_BLOCK

DATA_BLOCK "Clock_DB"   // DB50
// stored: AutoNumber false, InstanceOfName Clock, InstanceOfType FB
"Clock"
BEGIN
END_DATA_BLOCK

DATA_BLOCK "Com_DB"   // DB301
// stored: AutoNumber false, InstanceOfName Com, InstanceOfType FB
"Com"
BEGIN
END_DATA_BLOCK

DATA_BLOCK "DataTakeOver_DB"   // DB302
// stored: AutoNumber false, InstanceOfName DataTakeOver, InstanceOfType FB
"DataTakeOver"
BEGIN
END_DATA_BLOCK

DATA_BLOCK "Diag_DB"   // DB60
// stored: AutoNumber false, InstanceOfName Diag, InstanceOfType FB
"Diag"
BEGIN
END_DATA_BLOCK

DATA_BLOCK "ErrCom_DB"   // DB303
// stored: AutoNumber false, InstanceOfName ErrCom, InstanceOfType FB
"ErrCom"
BEGIN
END_DATA_BLOCK

DATA_BLOCK "Fault_DB"   // DB304
// stored: AutoNumber false, InstanceOfName Fault, InstanceOfType FB
"Fault"
BEGIN
END_DATA_BLOCK

DATA_BLOCK "SafetyCom_DB"   // DB45
// stored: AutoNumber false, InstanceOfName SafetyCom, InstanceOfType FB
"SafetyCom"
BEGIN
END_DATA_BLOCK

DATA_BLOCK "Sensors_DB"   // DB505
// stored: AutoNumber false, InstanceOfName Sensors, InstanceOfType FB
"Sensors"
BEGIN
END_DATA_BLOCK

DATA_BLOCK "TestIo_DB"   // DB306
// stored: AutoNumber false, InstanceOfName TestIo, InstanceOfType FB
"TestIo"
BEGIN
END_DATA_BLOCK
